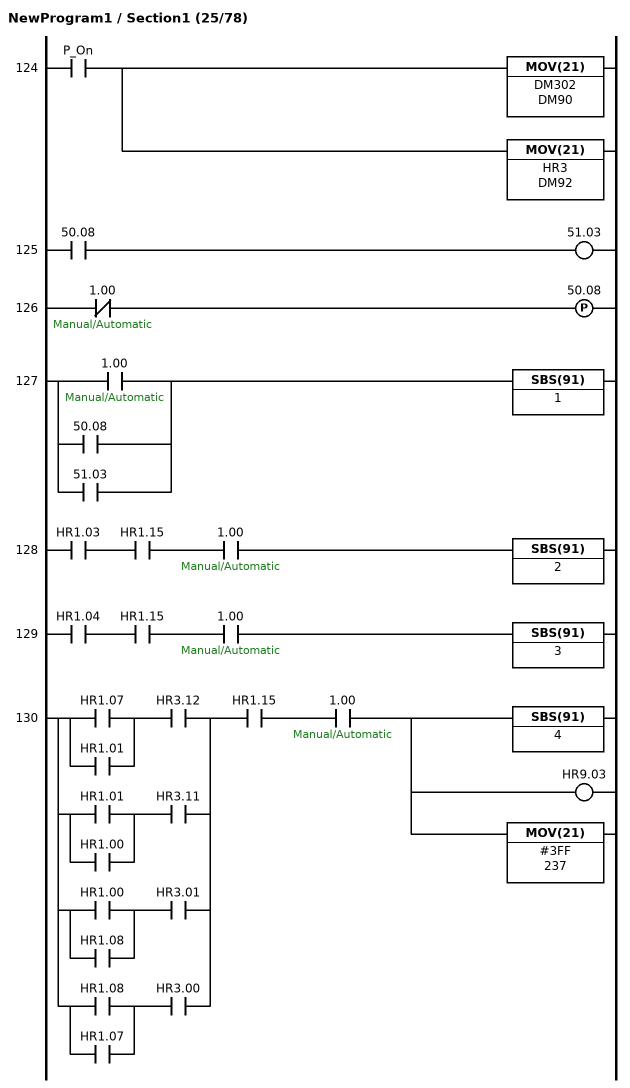
; [picture p24: NewProgram1 / Section1, rungs 124-130]
; rung 124
LD P_On
MOV(21) DM302 DM90
MOV(21) HR3 DM92
; rung 125
LD 50.08
OUT 51.03
; rung 126
LDNOT 1.00  ; Manual/Automatic
DIFU(13) 50.08
; rung 127
LD 1.00  ; Manual/Automatic
OR 50.08
OR 51.03
SBS(91) 1
; rung 128
LD HR1.03
AND HR1.15
AND 1.00  ; Manual/Automatic
SBS(91) 2
; rung 129
LD HR1.04
AND HR1.15
AND 1.00  ; Manual/Automatic
SBS(91) 3
; rung 130
LD HR1.07
OR HR1.01
AND HR3.12
LD HR1.01
OR HR1.00
AND HR3.11
ORLD
LD HR1.00
OR HR1.08
AND HR3.01
ORLD
LD HR1.08
OR HR1.07
AND HR3.00
ORLD
AND HR1.15
AND 1.00  ; Manual/Automatic
SBS(91) 4
OUT HR9.03
MOV(21) #3FF 237

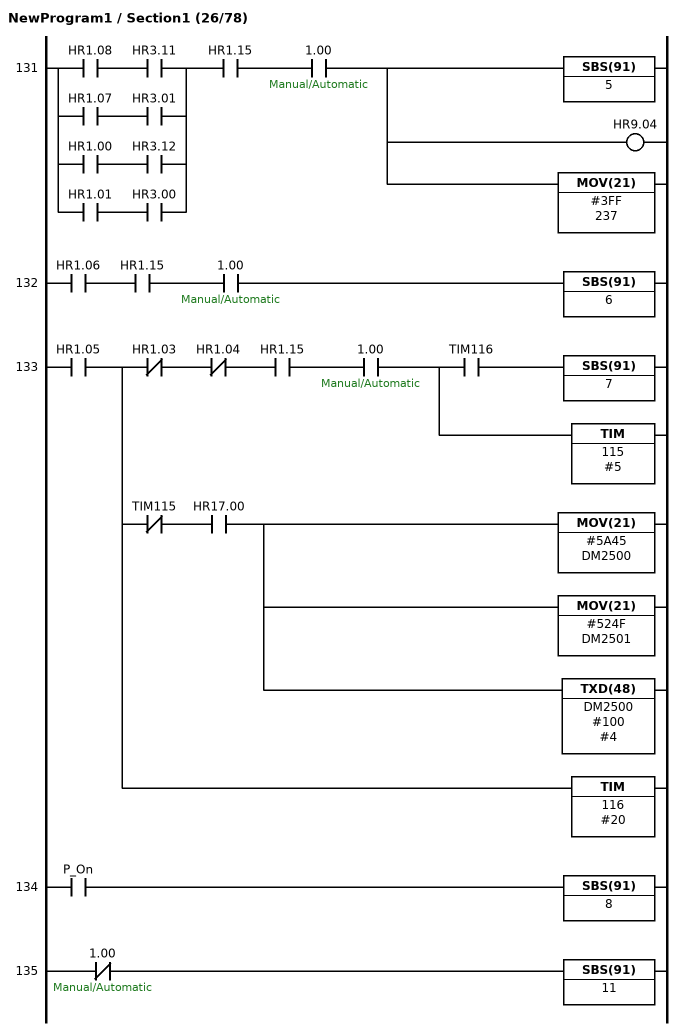
; rung 131
LD HR1.08
AND HR3.11
LD HR1.07
AND HR3.01
ORLD
LD HR1.00
AND HR3.12
ORLD
LD HR1.01
AND HR3.00
ORLD
AND HR1.15
AND 1.00  ; Manual/Automatic
SBS(91) 5
OUT HR9.04
MOV(21) #3FF 237
; rung 132
LD HR1.06
AND HR1.15
AND 1.00  ; Manual/Automatic
SBS(91) 6
; rung 133
LD HR1.05
OUT TR0
ANDNOT HR1.03
ANDNOT HR1.04
AND HR1.15
AND 1.00  ; Manual/Automatic
OUT TR1
AND TIM116
SBS(91) 7
LD TR1
TIM 115 #5
LD TR0
ANDNOT TIM115
AND HR17.00
MOV(21) #5A45 DM2500
MOV(21) #524F DM2501
TXD(48) DM2500 #100 #4
LD TR0
TIM 116 #20
; rung 134
LD P_On
SBS(91) 8
; rung 135
LDNOT 1.00  ; Manual/Automatic
SBS(91) 11

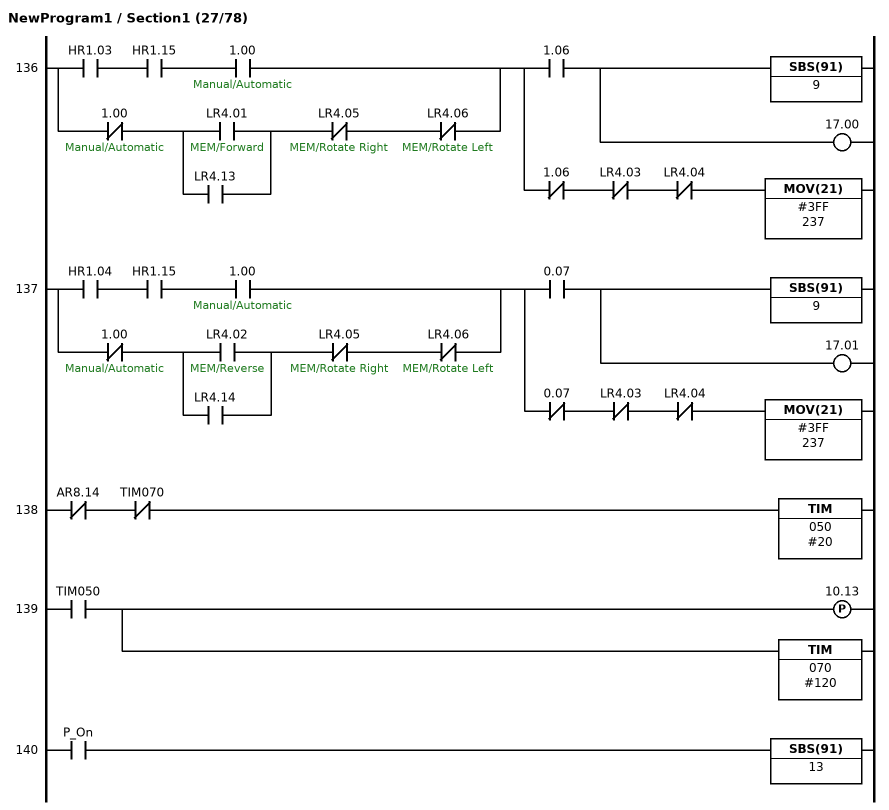
; rung 136
LD HR1.03
AND HR1.15
AND 1.00  ; Manual/Automatic
LDNOT 1.00  ; Manual/Automatic
LD LR4.01  ; MEM/Forward
OR LR4.13
ANDLD
ANDNOT LR4.05  ; MEM/Rotate Right
ANDNOT LR4.06  ; MEM/Rotate Left
ORLD
OUT TR0
AND 1.06
SBS(91) 9
OUT 17.00
LD TR0
ANDNOT 1.06
ANDNOT LR4.03
ANDNOT LR4.04
MOV(21) #3FF 237
; rung 137
LD HR1.04
AND HR1.15
AND 1.00  ; Manual/Automatic
LDNOT 1.00  ; Manual/Automatic
LD LR4.02  ; MEM/Reverse
OR LR4.14
ANDLD
ANDNOT LR4.05  ; MEM/Rotate Right
ANDNOT LR4.06  ; MEM/Rotate Left
ORLD
OUT TR0
AND 0.07
SBS(91) 9
OUT 17.01
LD TR0
ANDNOT 0.07
ANDNOT LR4.03
ANDNOT LR4.04
MOV(21) #3FF 237
; rung 138
LDNOT AR8.14
ANDNOT TIM070
TIM 050 #20
; rung 139
LD TIM050
DIFU(13) 10.13
TIM 070 #120
; rung 140
LD P_On
SBS(91) 13

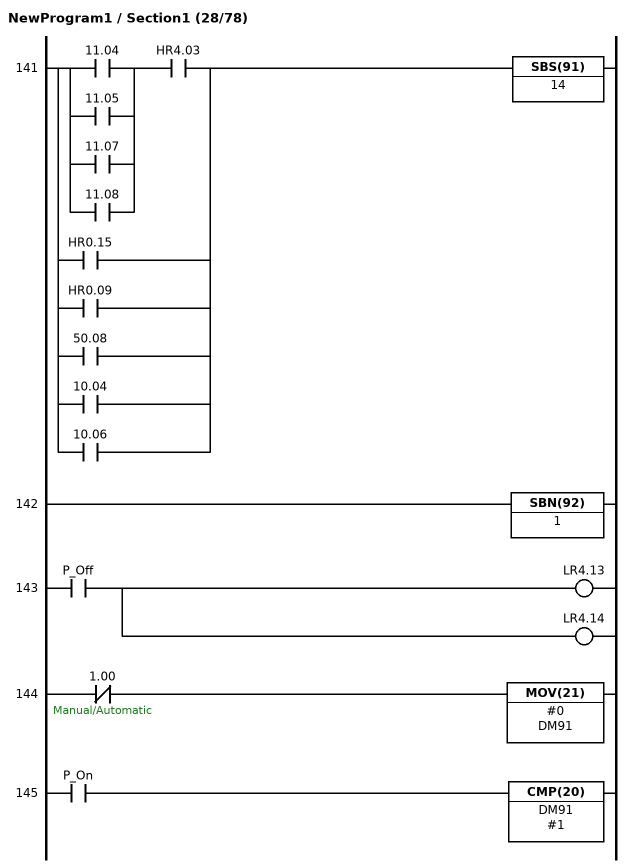
; rung 141
LD 11.04
OR 11.05
OR 11.07
OR 11.08
AND HR4.03
OR HR0.15
OR HR0.09
OR 50.08
OR 10.04
OR 10.06
SBS(91) 14
; rung 142
SBN(92) 1
; rung 143
LD P_Off
OUT LR4.13
OUT LR4.14
; rung 144
LDNOT 1.00  ; Manual/Automatic
MOV(21) #0 DM91
; rung 145
LD P_On
CMP(20) DM91 #1

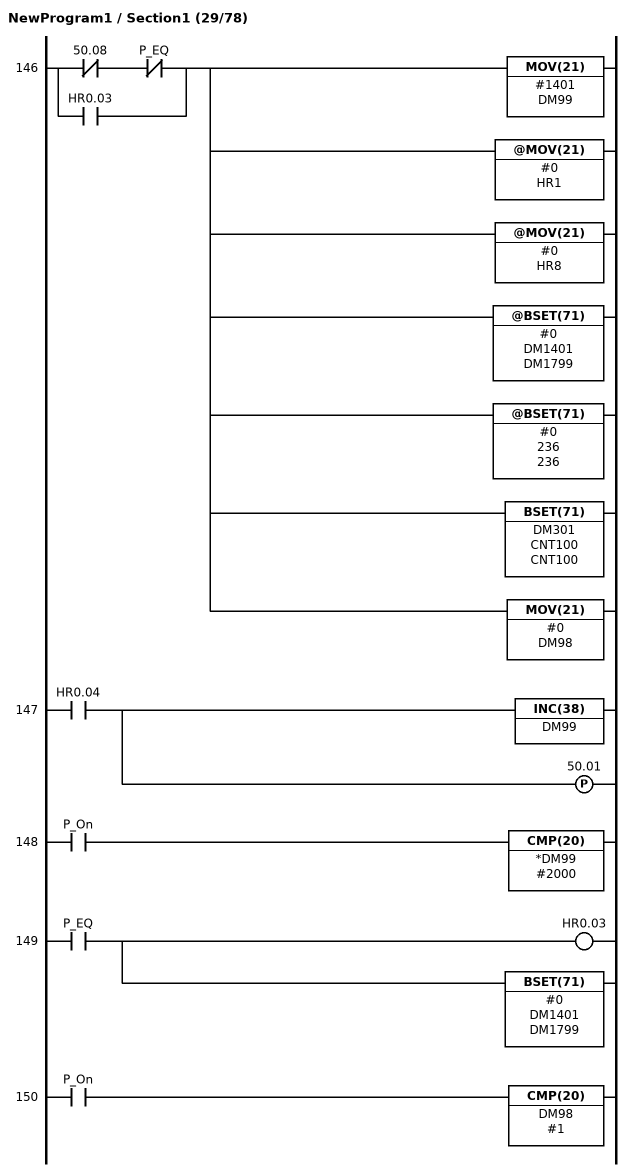
; rung 146
LDNOT 50.08
ANDNOT P_EQ
OR HR0.03
MOV(21) #1401 DM99
@MOV(21) #0 HR1
@MOV(21) #0 HR8
@BSET(71) #0 DM1401 DM1799
@BSET(71) #0 236 236
BSET(71) DM301 CNT100 CNT100
MOV(21) #0 DM98
; rung 147
LD HR0.04
INC(38) DM99
DIFU(13) 50.01
; rung 148
LD P_On
CMP(20) *DM99 #2000
; rung 149
LD P_EQ
OUT HR0.03
BSET(71) #0 DM1401 DM1799
; rung 150
LD P_On
CMP(20) DM98 #1

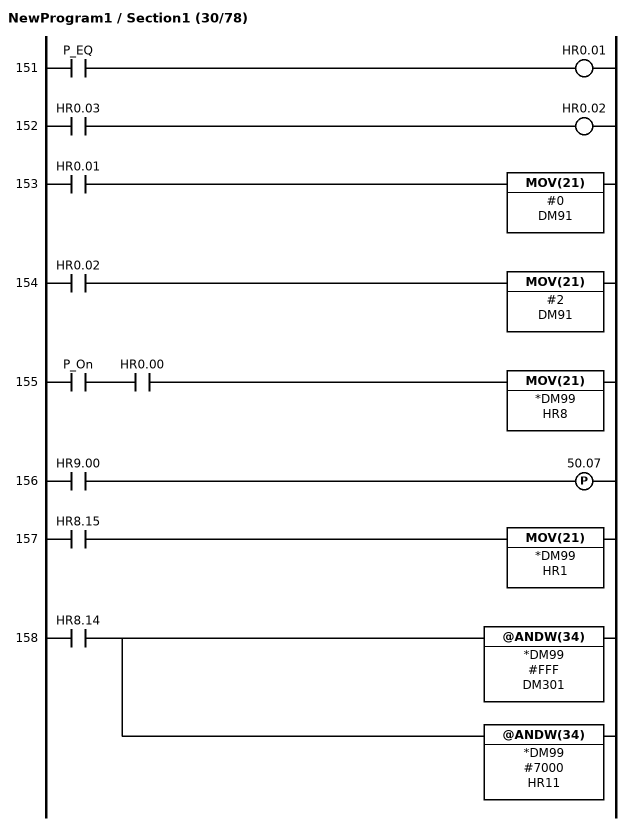
; rung 151
LD P_EQ
OUT HR0.01
; rung 152
LD HR0.03
OUT HR0.02
; rung 153
LD HR0.01
MOV(21) #0 DM91
; rung 154
LD HR0.02
MOV(21) #2 DM91
; rung 155
LD P_On
AND HR0.00
MOV(21) *DM99 HR8
; rung 156
LD HR9.00
DIFU(13) 50.07
; rung 157
LD HR8.15
MOV(21) *DM99 HR1
; rung 158
LD HR8.14
@ANDW(34) *DM99 #FFF DM301
@ANDW(34) *DM99 #7000 HR11

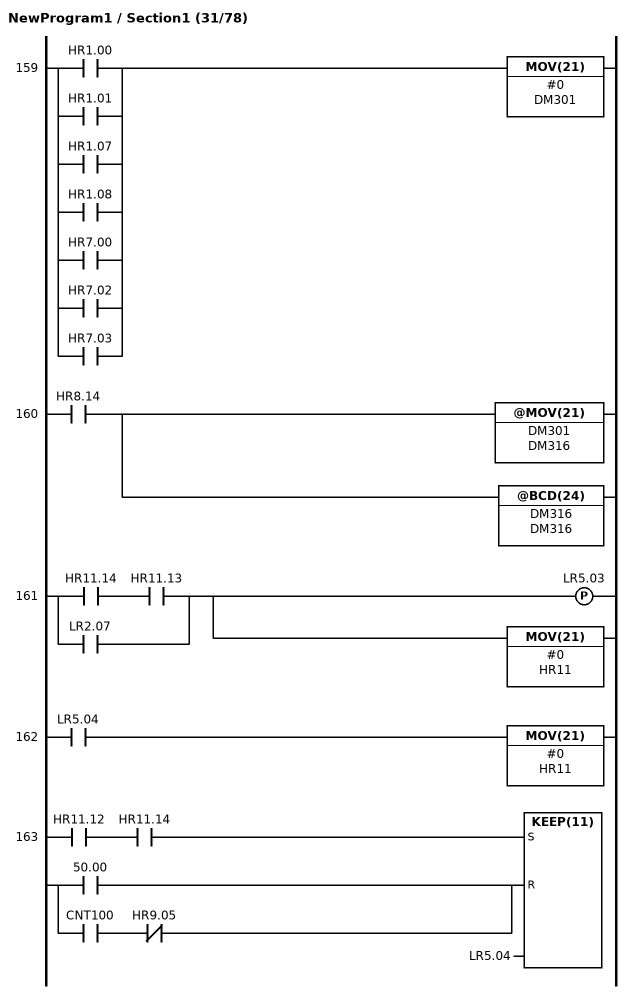
; rung 159
LD HR1.00
OR HR1.01
OR HR1.07
OR HR1.08
OR HR7.00
OR HR7.02
OR HR7.03
MOV(21) #0 DM301
; rung 160
LD HR8.14
@MOV(21) DM301 DM316
@BCD(24) DM316 DM316
; rung 161
LD HR11.14
AND HR11.13
OR LR2.07
DIFU(13) LR5.03
MOV(21) #0 HR11
; rung 162
LD LR5.04
MOV(21) #0 HR11
; rung 163
LD HR11.12
AND HR11.14
LD 50.00
LD CNT100
ANDNOT HR9.05
ORLD
KEEP(11) LR5.04

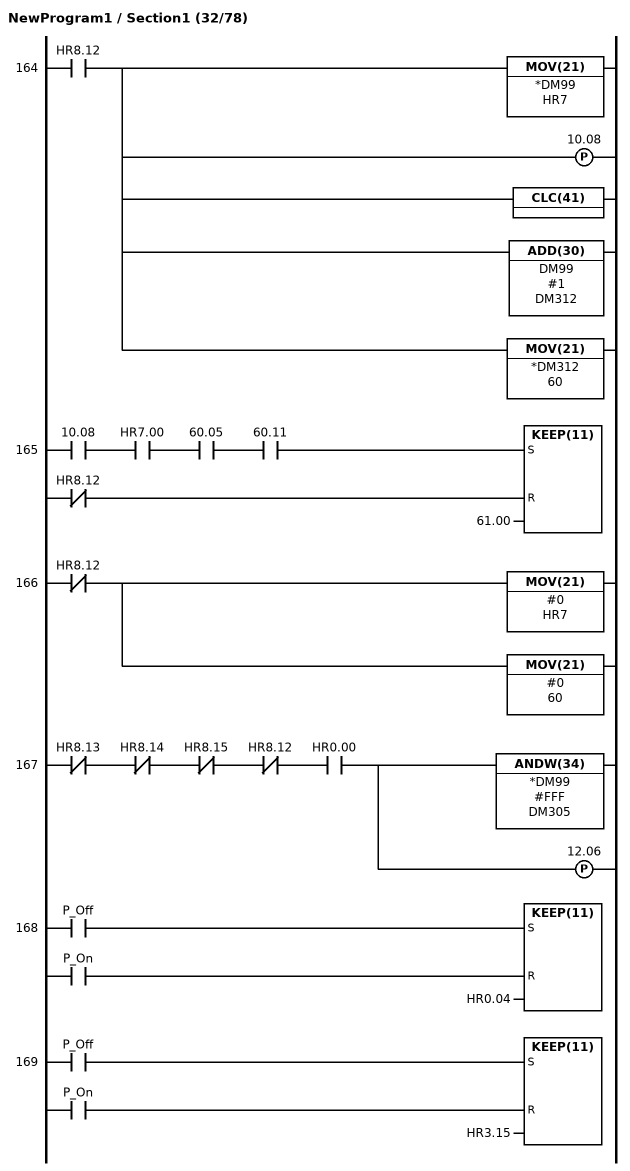
; rung 164
LD HR8.12
MOV(21) *DM99 HR7
DIFU(13) 10.08
CLC(41)
ADD(30) DM99 #1 DM312
MOV(21) *DM312 60
; rung 165
LD 10.08
AND HR7.00
AND 60.05
AND 60.11
LDNOT HR8.12
KEEP(11) 61.00
; rung 166
LDNOT HR8.12
MOV(21) #0 HR7
MOV(21) #0 60
; rung 167
LDNOT HR8.13
ANDNOT HR8.14
ANDNOT HR8.15
ANDNOT HR8.12
AND HR0.00
ANDW(34) *DM99 #FFF DM305
DIFU(13) 12.06
; rung 168
LD P_Off
LD P_On
KEEP(11) HR0.04
; rung 169
LD P_Off
LD P_On
KEEP(11) HR3.15

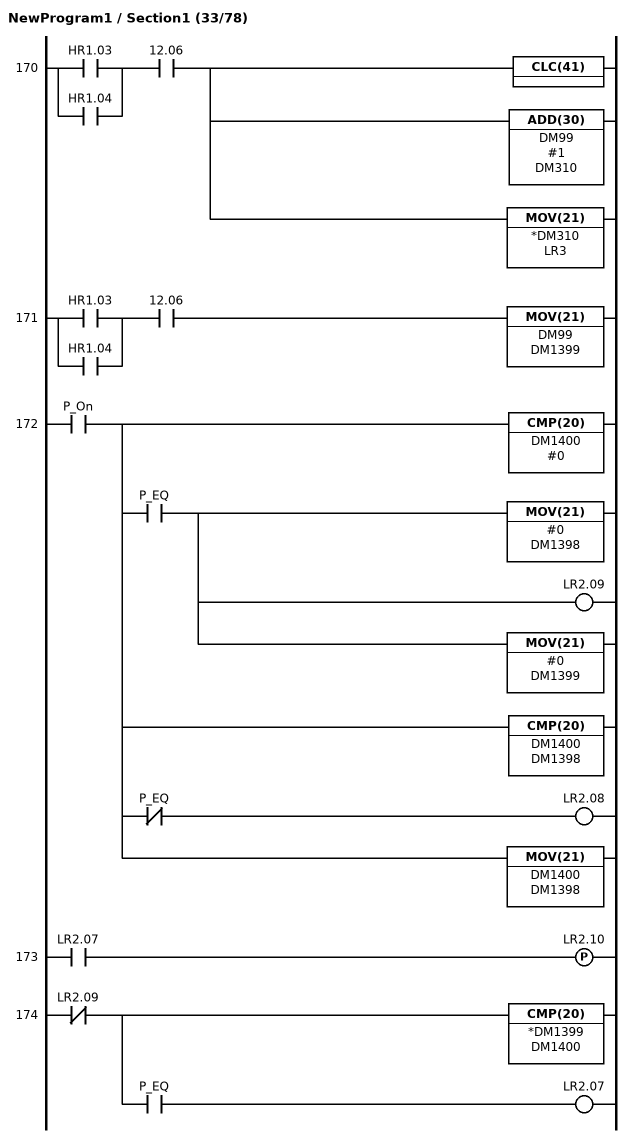
; rung 170
LD HR1.03
OR HR1.04
AND 12.06
CLC(41)
ADD(30) DM99 #1 DM310
MOV(21) *DM310 LR3
; rung 171
LD HR1.03
OR HR1.04
AND 12.06
MOV(21) DM99 DM1399
; rung 172
LD P_On
OUT TR0
CMP(20) DM1400 #0
AND P_EQ
MOV(21) #0 DM1398
OUT LR2.09
MOV(21) #0 DM1399
LD TR0
CMP(20) DM1400 DM1398
ANDNOT P_EQ
OUT LR2.08
LD TR0
MOV(21) DM1400 DM1398
; rung 173
LD LR2.07
DIFU(13) LR2.10
; rung 174
LDNOT LR2.09
CMP(20) *DM1399 DM1400
AND P_EQ
OUT LR2.07

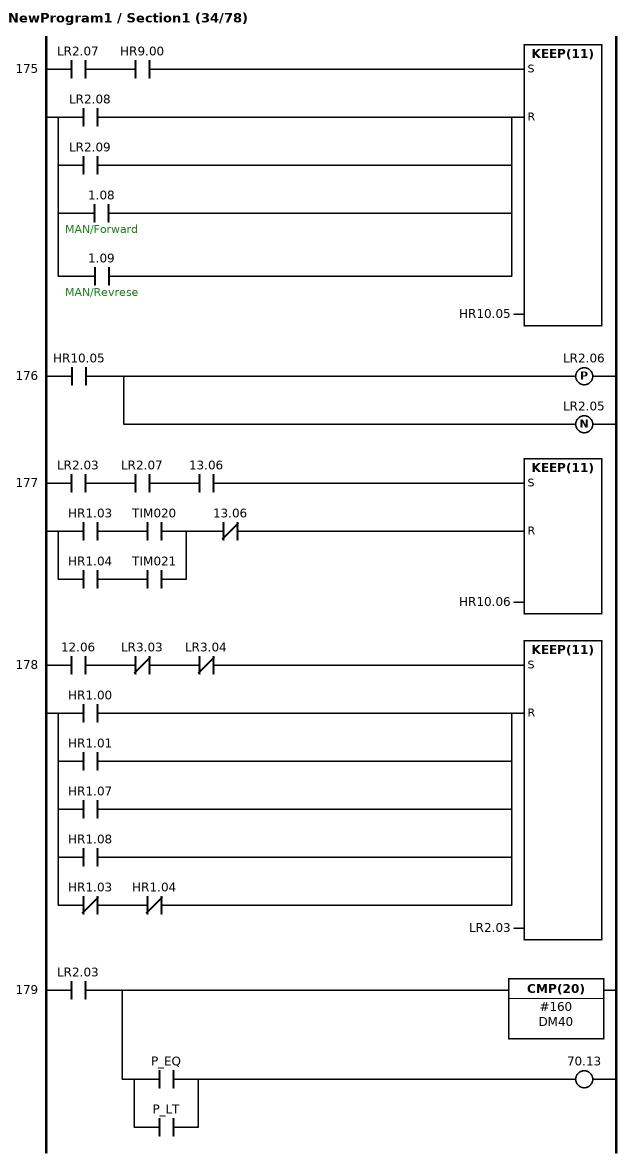
; rung 175
LD LR2.07
AND HR9.00
LD LR2.08
OR LR2.09
OR 1.08  ; MAN/Forward
OR 1.09  ; MAN/Revrese
KEEP(11) HR10.05
; rung 176
LD HR10.05
DIFU(13) LR2.06
DIFD(14) LR2.05
; rung 177
LD LR2.03
AND LR2.07
AND 13.06
LD HR1.03
AND TIM020
LD HR1.04
AND TIM021
ORLD
ANDNOT 13.06
KEEP(11) HR10.06
; rung 178
LD 12.06
ANDNOT LR3.03
ANDNOT LR3.04
LD HR1.00
OR HR1.01
OR HR1.07
OR HR1.08
LDNOT HR1.03
ANDNOT HR1.04
ORLD
KEEP(11) LR2.03
; rung 179
LD LR2.03
CMP(20) #160 DM40
LD P_EQ
OR P_LT
ANDLD
OUT 70.13

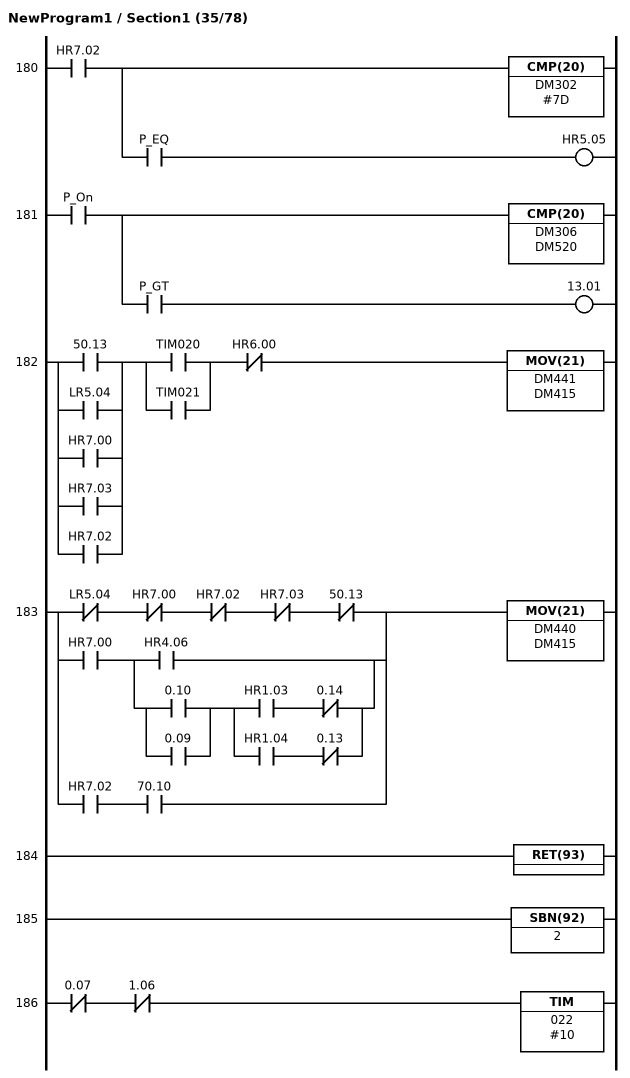
; rung 180
LD HR7.02
CMP(20) DM302 #7D
AND P_EQ
OUT HR5.05
; rung 181
LD P_On
CMP(20) DM306 DM520
AND P_GT
OUT 13.01
; rung 182
LD 50.13
OR LR5.04
OR HR7.00
OR HR7.03
OR HR7.02
LD TIM020
OR TIM021
ANDLD
ANDNOT HR6.00
MOV(21) DM441 DM415
; rung 183
LDNOT LR5.04
ANDNOT HR7.00
ANDNOT HR7.02
ANDNOT HR7.03
ANDNOT 50.13
LD HR7.00
LD HR4.06
LD 0.10
OR 0.09
LD HR1.03
ANDNOT 0.14
LD HR1.04
ANDNOT 0.13
ORLD
ANDLD
ORLD
ANDLD
ORLD
LD HR7.02
AND 70.10
ORLD
MOV(21) DM440 DM415
; rung 184
RET(93)
; rung 185
SBN(92) 2
; rung 186
LDNOT 0.07
ANDNOT 1.06
TIM 022 #10

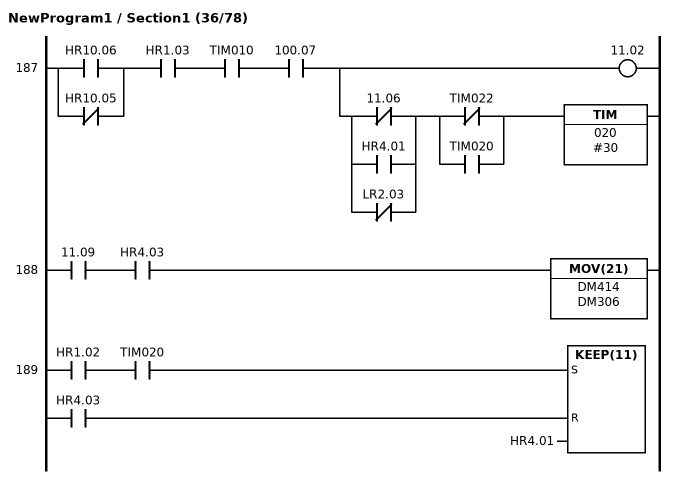
; rung 187
LD HR10.06
ORNOT HR10.05
AND HR1.03
AND TIM010
AND 100.07
OUT 11.02
LDNOT 11.06
OR HR4.01
ORNOT LR2.03
ANDLD
LDNOT TIM022
OR TIM020
ANDLD
TIM 020 #30
; rung 188
LD 11.09
AND HR4.03
MOV(21) DM414 DM306
; rung 189
LD HR1.02
AND TIM020
LD HR4.03
KEEP(11) HR4.01

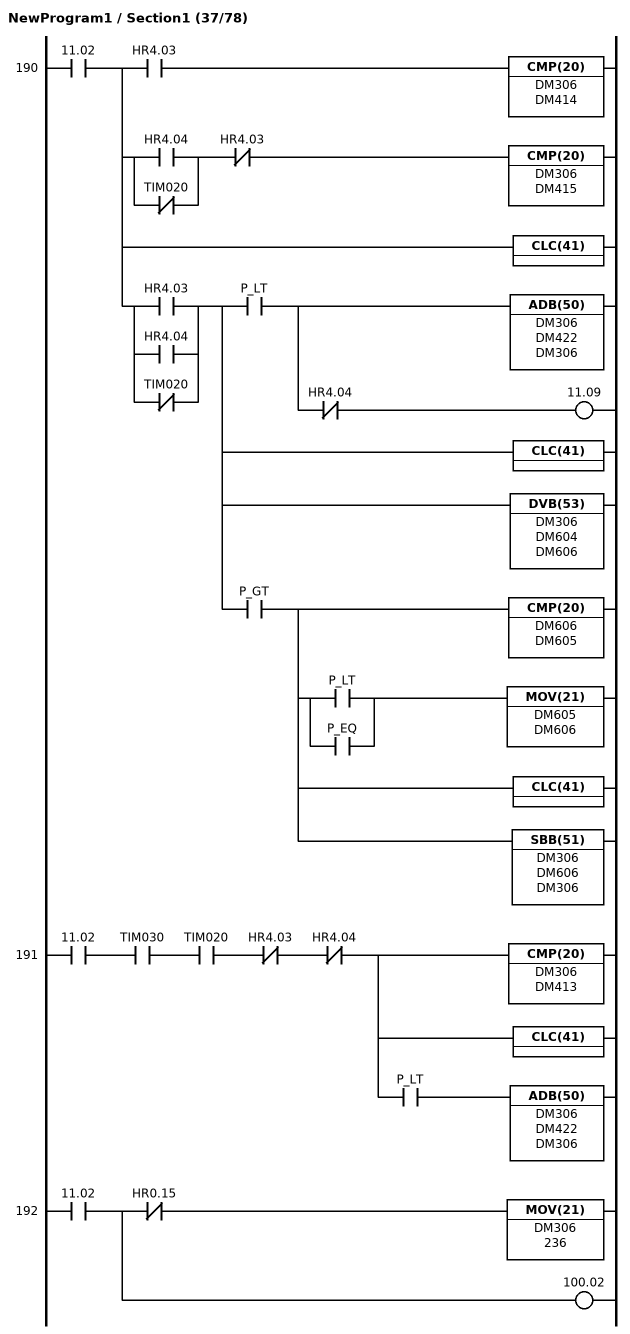
; rung 190
LD 11.02
OUT TR0
AND HR4.03
CMP(20) DM306 DM414
LD TR0
LD HR4.04
ORNOT TIM020
ANDLD
ANDNOT HR4.03
CMP(20) DM306 DM415
LD TR0
CLC(41)
LD HR4.03
OR HR4.04
ORNOT TIM020
ANDLD
OUT TR0
AND P_LT
ADB(50) DM306 DM422 DM306
ANDNOT HR4.04
OUT 11.09
LD TR0
CLC(41)
DVB(53) DM306 DM604 DM606
AND P_GT
OUT TR0
CMP(20) DM606 DM605
LD P_LT
OR P_EQ
ANDLD
MOV(21) DM605 DM606
LD TR0
CLC(41)
SBB(51) DM306 DM606 DM306
; rung 191
LD 11.02
AND TIM030
AND TIM020
ANDNOT HR4.03
ANDNOT HR4.04
CMP(20) DM306 DM413
CLC(41)
AND P_LT
ADB(50) DM306 DM422 DM306
; rung 192
LD 11.02
OUT TR0
ANDNOT HR0.15
MOV(21) DM306 236
LD TR0
OUT 100.02

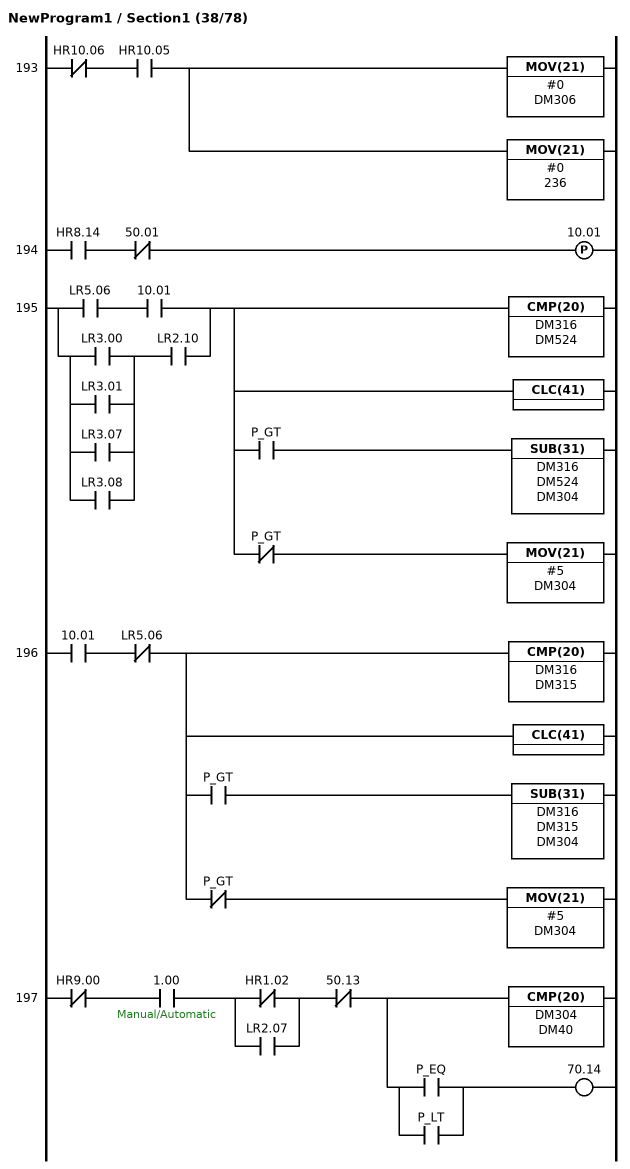
; rung 193
LDNOT HR10.06
AND HR10.05
MOV(21) #0 DM306
MOV(21) #0 236
; rung 194
LD HR8.14
ANDNOT 50.01
DIFU(13) 10.01
; rung 195
LD LR5.06
AND 10.01
LD LR3.00
OR LR3.01
OR LR3.07
OR LR3.08
AND LR2.10
ORLD
OUT TR0
CMP(20) DM316 DM524
CLC(41)
AND P_GT
SUB(31) DM316 DM524 DM304
LD TR0
ANDNOT P_GT
MOV(21) #5 DM304
; rung 196
LD 10.01
ANDNOT LR5.06
OUT TR0
CMP(20) DM316 DM315
CLC(41)
AND P_GT
SUB(31) DM316 DM315 DM304
LD TR0
ANDNOT P_GT
MOV(21) #5 DM304
; rung 197
LDNOT HR9.00
AND 1.00  ; Manual/Automatic
LDNOT HR1.02
OR LR2.07
ANDLD
ANDNOT 50.13
CMP(20) DM304 DM40
LD P_EQ
OR P_LT
ANDLD
OUT 70.14

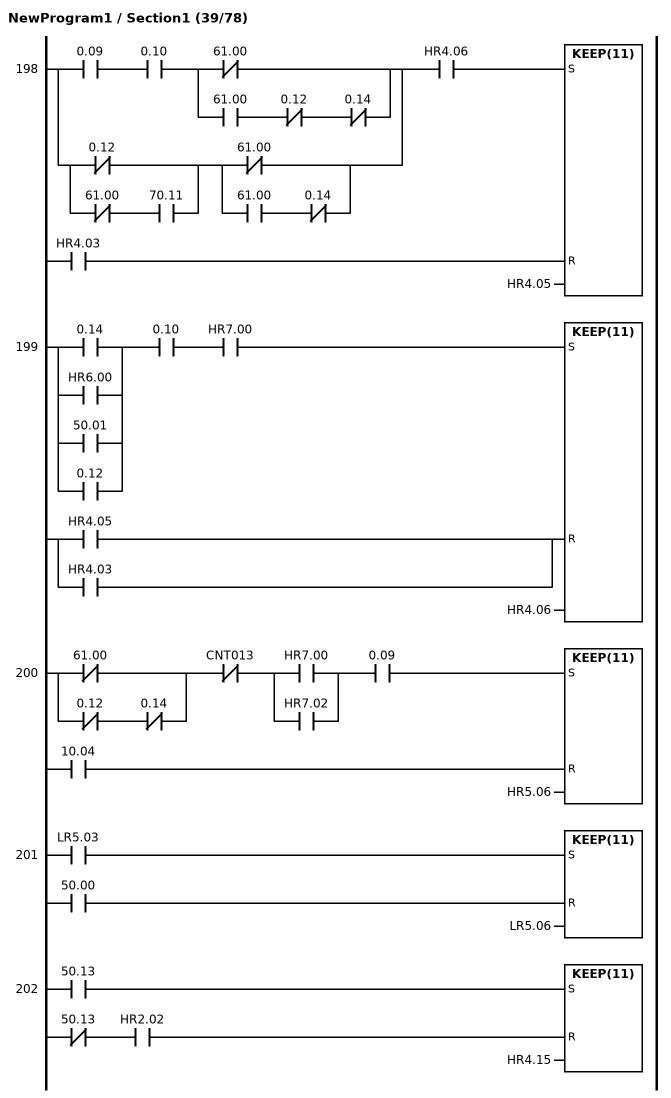
; rung 198
LD 0.09
AND 0.10
LDNOT 61.00
LD 61.00
ANDNOT 0.12
ANDNOT 0.14
ORLD
ANDLD
LDNOT 0.12
LDNOT 61.00
AND 70.11
ORLD
LDNOT 61.00
LD 61.00
ANDNOT 0.14
ORLD
ANDLD
ORLD
AND HR4.06
LD HR4.03
KEEP(11) HR4.05
; rung 199
LD 0.14
OR HR6.00
OR 50.01
OR 0.12
AND 0.10
AND HR7.00
LD HR4.05
OR HR4.03
KEEP(11) HR4.06
; rung 200
LDNOT 61.00
LDNOT 0.12
ANDNOT 0.14
ORLD
ANDNOT CNT013
LD HR7.00
OR HR7.02
ANDLD
AND 0.09
LD 10.04
KEEP(11) HR5.06
; rung 201
LD LR5.03
LD 50.00
KEEP(11) LR5.06
; rung 202
LD 50.13
LDNOT 50.13
AND HR2.02
KEEP(11) HR4.15

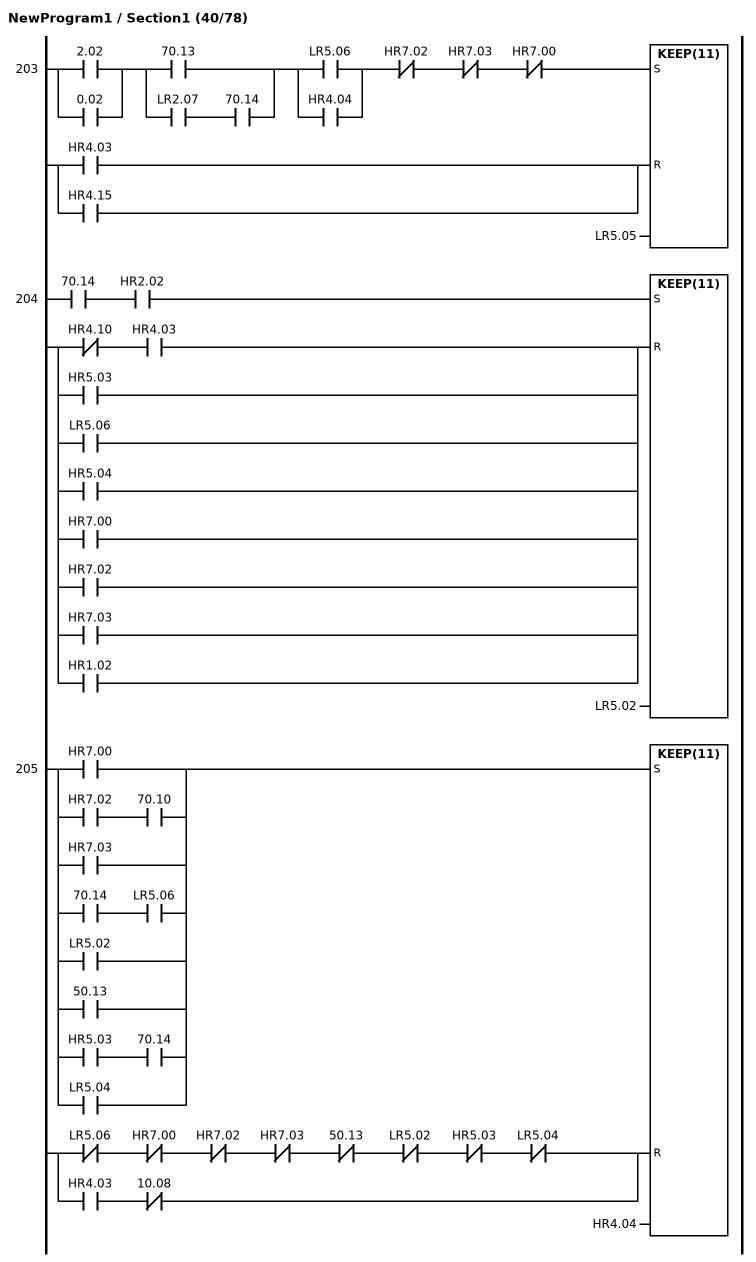
; rung 203
LD 2.02
OR 0.02
LD 70.13
LD LR2.07
AND 70.14
ORLD
ANDLD
LD LR5.06
OR HR4.04
ANDLD
ANDNOT HR7.02
ANDNOT HR7.03
ANDNOT HR7.00
LD HR4.03
OR HR4.15
KEEP(11) LR5.05
; rung 204
LD 70.14
AND HR2.02
LDNOT HR4.10
AND HR4.03
OR HR5.03
OR LR5.06
OR HR5.04
OR HR7.00
OR HR7.02
OR HR7.03
OR HR1.02
KEEP(11) LR5.02
; rung 205
LD HR7.00
LD HR7.02
AND 70.10
ORLD
OR HR7.03
LD 70.14
AND LR5.06
ORLD
OR LR5.02
OR 50.13
LD HR5.03
AND 70.14
ORLD
OR LR5.04
LDNOT LR5.06
ANDNOT HR7.00
ANDNOT HR7.02
ANDNOT HR7.03
ANDNOT 50.13
ANDNOT LR5.02
ANDNOT HR5.03
ANDNOT LR5.04
LD HR4.03
ANDNOT 10.08
ORLD
KEEP(11) HR4.04

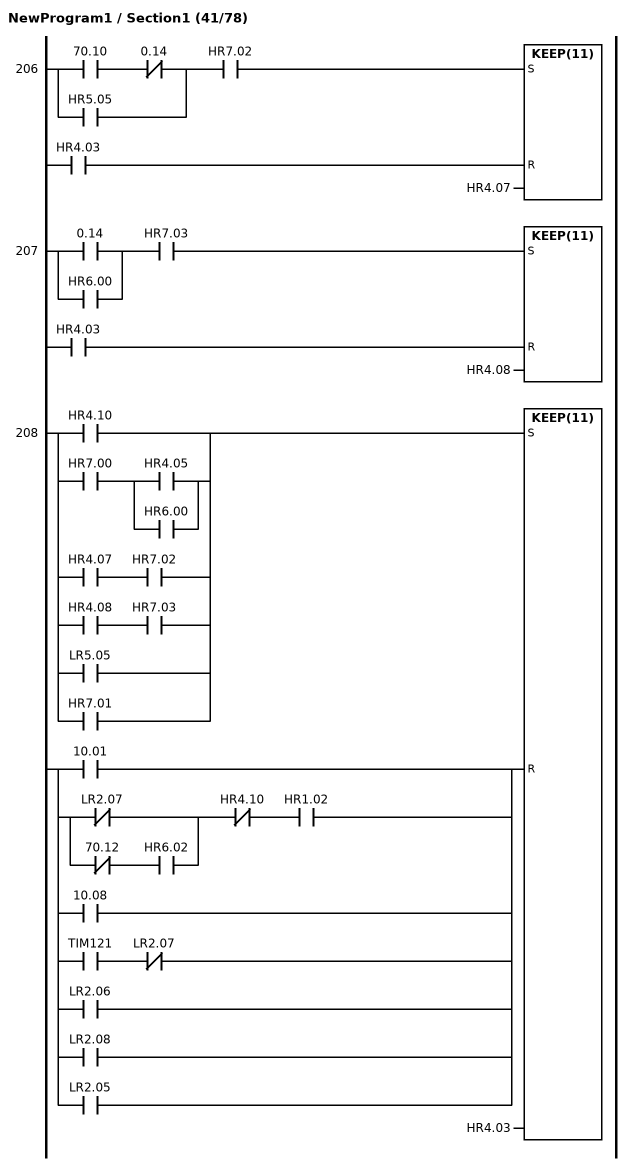
; rung 206
LD 70.10
ANDNOT 0.14
OR HR5.05
AND HR7.02
LD HR4.03
KEEP(11) HR4.07
; rung 207
LD 0.14
OR HR6.00
AND HR7.03
LD HR4.03
KEEP(11) HR4.08
; rung 208
LD HR4.10
LD HR7.00
LD HR4.05
OR HR6.00
ANDLD
ORLD
LD HR4.07
AND HR7.02
ORLD
LD HR4.08
AND HR7.03
ORLD
OR LR5.05
OR HR7.01
LD 10.01
LDNOT LR2.07
LDNOT 70.12
AND HR6.02
ORLD
ANDNOT HR4.10
AND HR1.02
ORLD
OR 10.08
LD TIM121
ANDNOT LR2.07
ORLD
OR LR2.06
OR LR2.08
OR LR2.05
KEEP(11) HR4.03

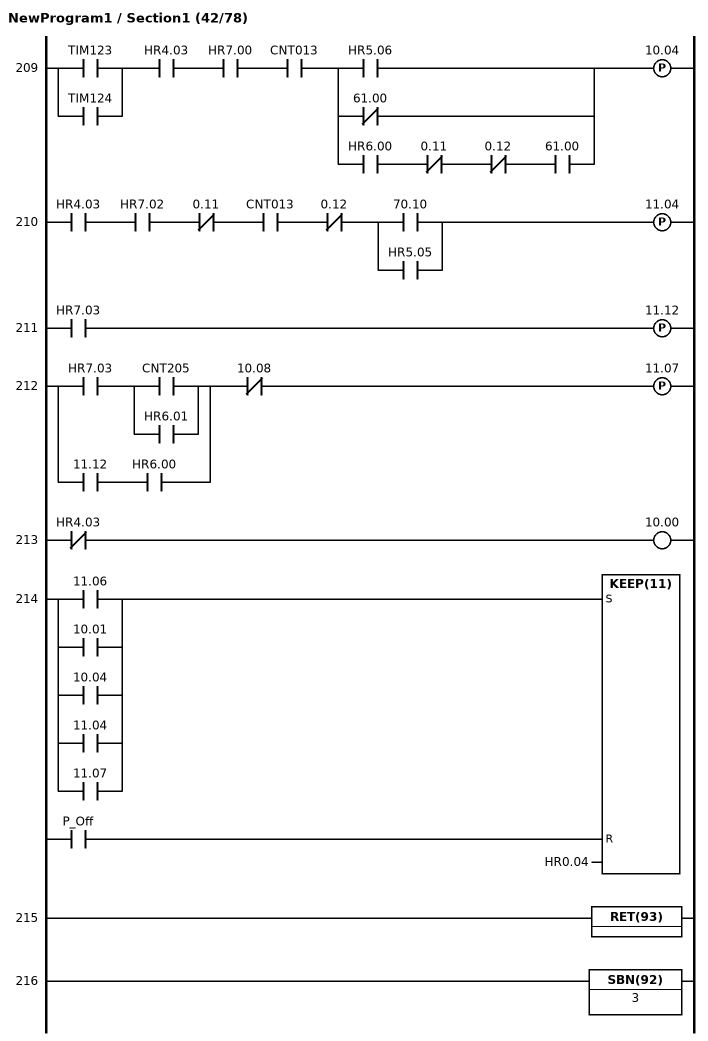
; rung 209
LD TIM123
OR TIM124
AND HR4.03
AND HR7.00
AND CNT013
LD HR5.06
ORNOT 61.00
LD HR6.00
ANDNOT 0.11
ANDNOT 0.12
AND 61.00
ORLD
ANDLD
DIFU(13) 10.04
; rung 210
LD HR4.03
AND HR7.02
ANDNOT 0.11
AND CNT013
ANDNOT 0.12
LD 70.10
OR HR5.05
ANDLD
DIFU(13) 11.04
; rung 211
LD HR7.03
DIFU(13) 11.12
; rung 212
LD HR7.03
LD CNT205
OR HR6.01
ANDLD
LD 11.12
AND HR6.00
ORLD
ANDNOT 10.08
DIFU(13) 11.07
; rung 213
LDNOT HR4.03
OUT 10.00
; rung 214
LD 11.06
OR 10.01
OR 10.04
OR 11.04
OR 11.07
LD P_Off
KEEP(11) HR0.04
; rung 215
RET(93)
; rung 216
SBN(92) 3

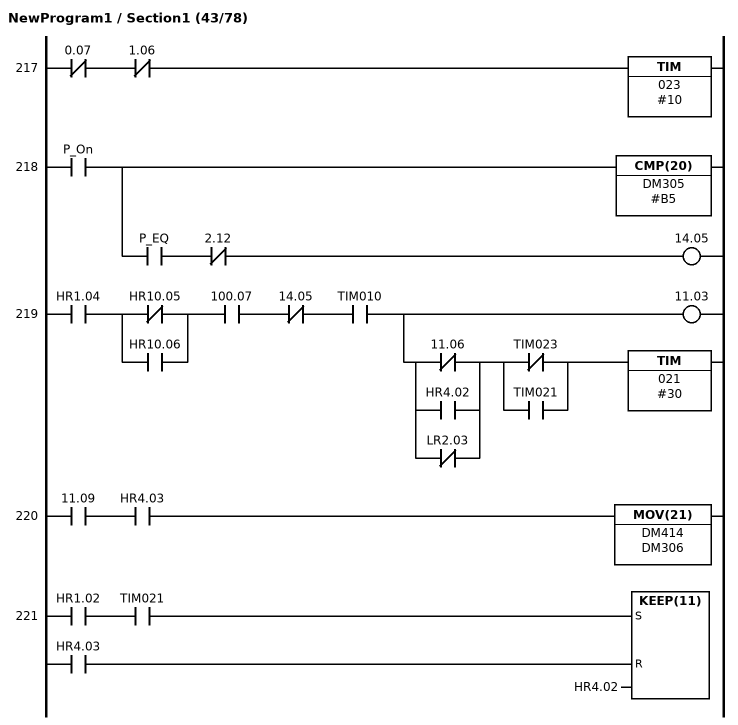
; rung 217
LDNOT 0.07
ANDNOT 1.06
TIM 023 #10
; rung 218
LD P_On
CMP(20) DM305 #B5
AND P_EQ
ANDNOT 2.12
OUT 14.05
; rung 219
LD HR1.04
LDNOT HR10.05
OR HR10.06
ANDLD
AND 100.07
ANDNOT 14.05
AND TIM010
OUT 11.03
LDNOT 11.06
OR HR4.02
ORNOT LR2.03
ANDLD
LDNOT TIM023
OR TIM021
ANDLD
TIM 021 #30
; rung 220
LD 11.09
AND HR4.03
MOV(21) DM414 DM306
; rung 221
LD HR1.02
AND TIM021
LD HR4.03
KEEP(11) HR4.02

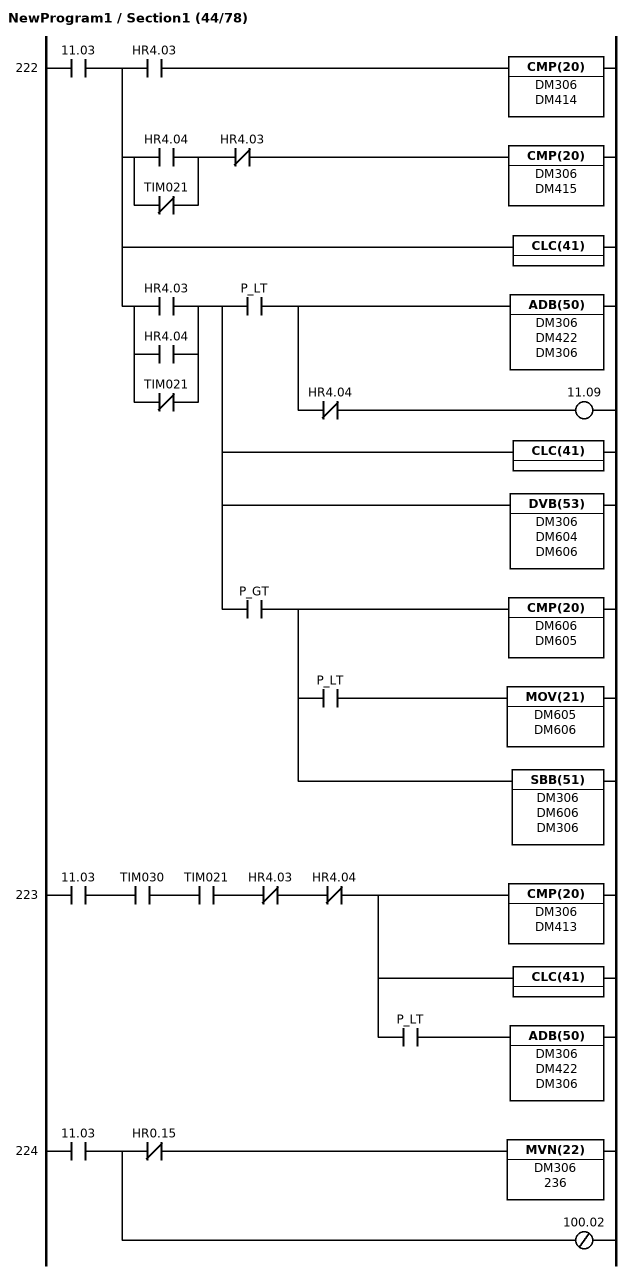
; rung 222
LD 11.03
OUT TR0
AND HR4.03
CMP(20) DM306 DM414
LD TR0
LD HR4.04
ORNOT TIM021
ANDLD
ANDNOT HR4.03
CMP(20) DM306 DM415
LD TR0
CLC(41)
LD HR4.03
OR HR4.04
ORNOT TIM021
ANDLD
OUT TR0
AND P_LT
ADB(50) DM306 DM422 DM306
ANDNOT HR4.04
OUT 11.09
LD TR0
CLC(41)
DVB(53) DM306 DM604 DM606
AND P_GT
OUT TR0
CMP(20) DM606 DM605
AND P_LT
MOV(21) DM605 DM606
LD TR0
SBB(51) DM306 DM606 DM306
; rung 223
LD 11.03
AND TIM030
AND TIM021
ANDNOT HR4.03
ANDNOT HR4.04
CMP(20) DM306 DM413
CLC(41)
AND P_LT
ADB(50) DM306 DM422 DM306
; rung 224
LD 11.03
OUT TR0
ANDNOT HR0.15
MVN(22) DM306 236
LD TR0
OUTNOT 100.02

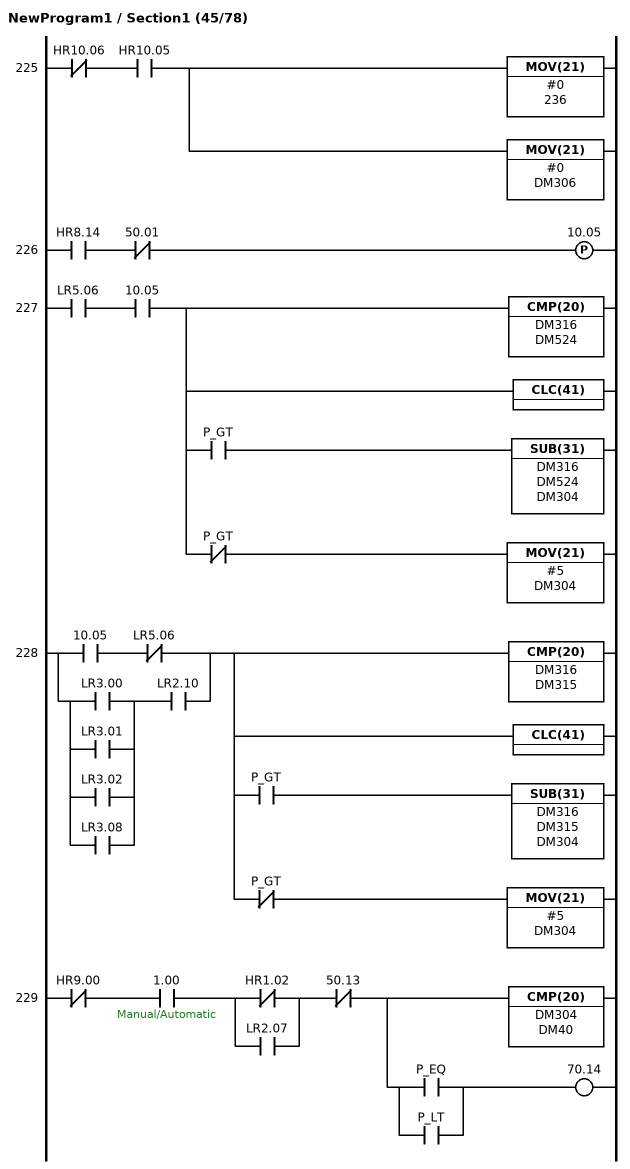
; rung 225
LDNOT HR10.06
AND HR10.05
MOV(21) #0 236
MOV(21) #0 DM306
; rung 226
LD HR8.14
ANDNOT 50.01
DIFU(13) 10.05
; rung 227
LD LR5.06
AND 10.05
OUT TR0
CMP(20) DM316 DM524
CLC(41)
AND P_GT
SUB(31) DM316 DM524 DM304
LD TR0
ANDNOT P_GT
MOV(21) #5 DM304
; rung 228
LD 10.05
ANDNOT LR5.06
LD LR3.00
OR LR3.01
OR LR3.02
OR LR3.08
AND LR2.10
ORLD
OUT TR0
CMP(20) DM316 DM315
CLC(41)
AND P_GT
SUB(31) DM316 DM315 DM304
LD TR0
ANDNOT P_GT
MOV(21) #5 DM304
; rung 229
LDNOT HR9.00
AND 1.00  ; Manual/Automatic
LDNOT HR1.02
OR LR2.07
ANDLD
ANDNOT 50.13
CMP(20) DM304 DM40
LD P_EQ
OR P_LT
ANDLD
OUT 70.14

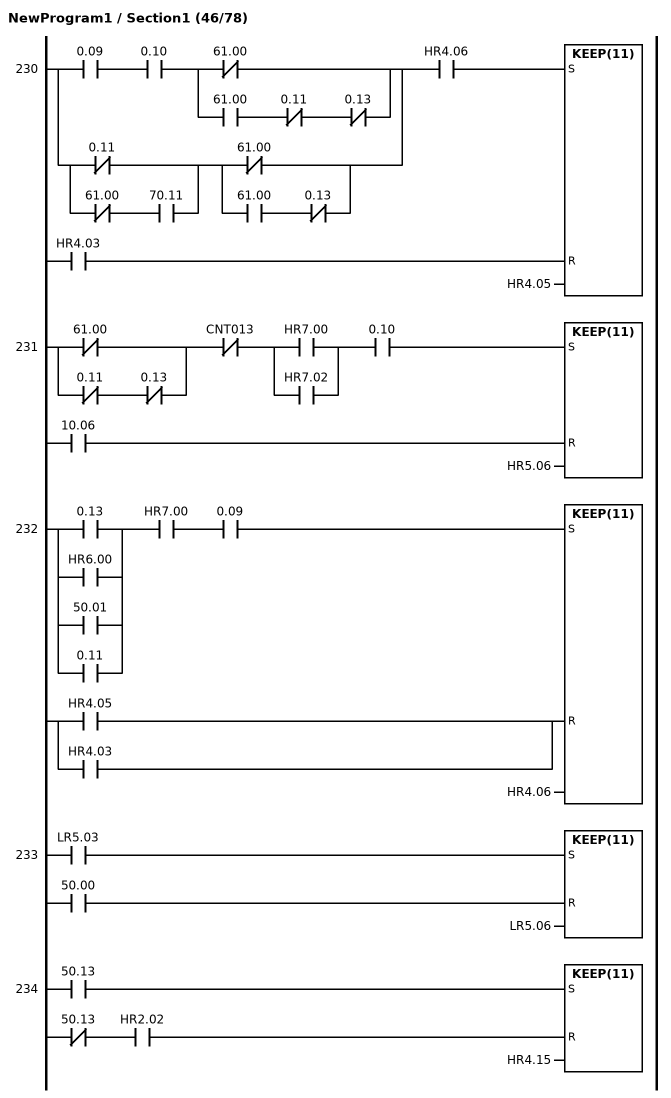
; rung 230
LD 0.09
AND 0.10
LDNOT 61.00
LD 61.00
ANDNOT 0.11
ANDNOT 0.13
ORLD
ANDLD
LDNOT 0.11
LDNOT 61.00
AND 70.11
ORLD
LDNOT 61.00
LD 61.00
ANDNOT 0.13
ORLD
ANDLD
ORLD
AND HR4.06
LD HR4.03
KEEP(11) HR4.05
; rung 231
LDNOT 61.00
LDNOT 0.11
ANDNOT 0.13
ORLD
ANDNOT CNT013
LD HR7.00
OR HR7.02
ANDLD
AND 0.10
LD 10.06
KEEP(11) HR5.06
; rung 232
LD 0.13
OR HR6.00
OR 50.01
OR 0.11
AND HR7.00
AND 0.09
LD HR4.05
OR HR4.03
KEEP(11) HR4.06
; rung 233
LD LR5.03
LD 50.00
KEEP(11) LR5.06
; rung 234
LD 50.13
LDNOT 50.13
AND HR2.02
KEEP(11) HR4.15

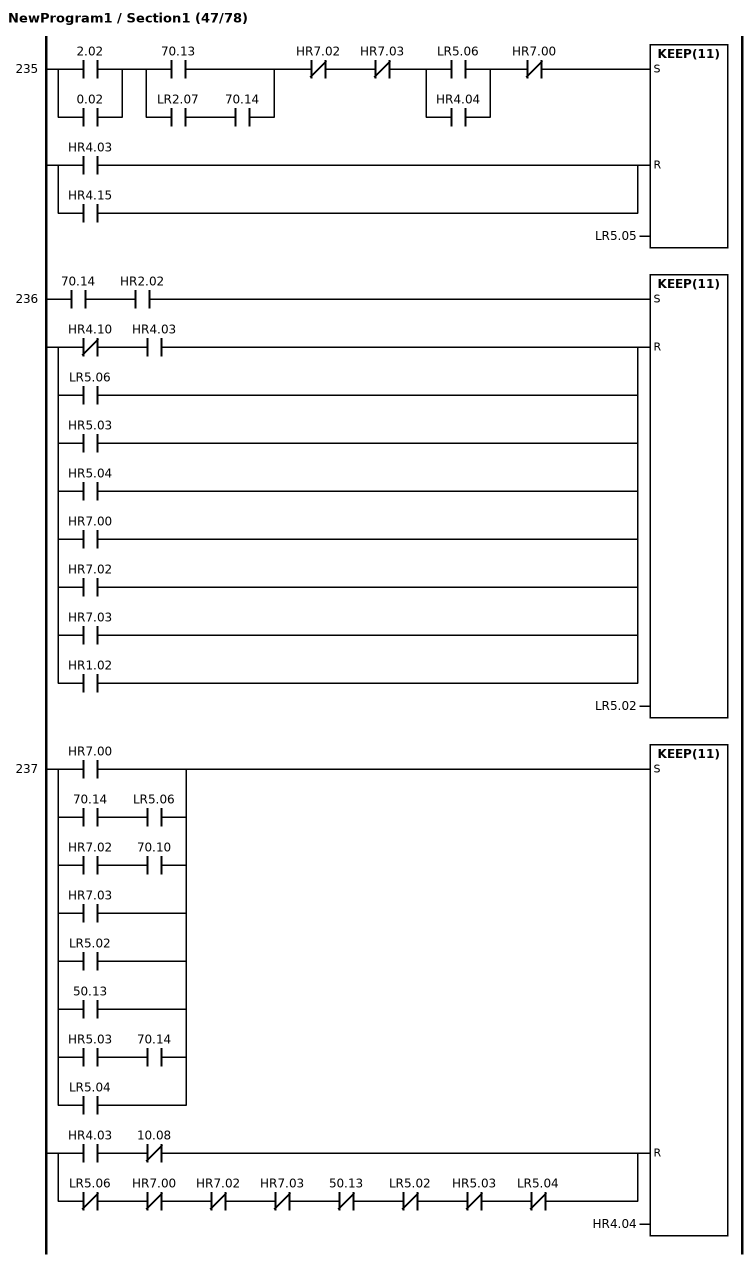
; rung 235
LD 2.02
OR 0.02
LD 70.13
LD LR2.07
AND 70.14
ORLD
ANDLD
ANDNOT HR7.02
ANDNOT HR7.03
LD LR5.06
OR HR4.04
ANDLD
ANDNOT HR7.00
LD HR4.03
OR HR4.15
KEEP(11) LR5.05
; rung 236
LD 70.14
AND HR2.02
LDNOT HR4.10
AND HR4.03
OR LR5.06
OR HR5.03
OR HR5.04
OR HR7.00
OR HR7.02
OR HR7.03
OR HR1.02
KEEP(11) LR5.02
; rung 237
LD HR7.00
LD 70.14
AND LR5.06
ORLD
LD HR7.02
AND 70.10
ORLD
OR HR7.03
OR LR5.02
OR 50.13
LD HR5.03
AND 70.14
ORLD
OR LR5.04
LD HR4.03
ANDNOT 10.08
LDNOT LR5.06
ANDNOT HR7.00
ANDNOT HR7.02
ANDNOT HR7.03
ANDNOT 50.13
ANDNOT LR5.02
ANDNOT HR5.03
ANDNOT LR5.04
ORLD
KEEP(11) HR4.04

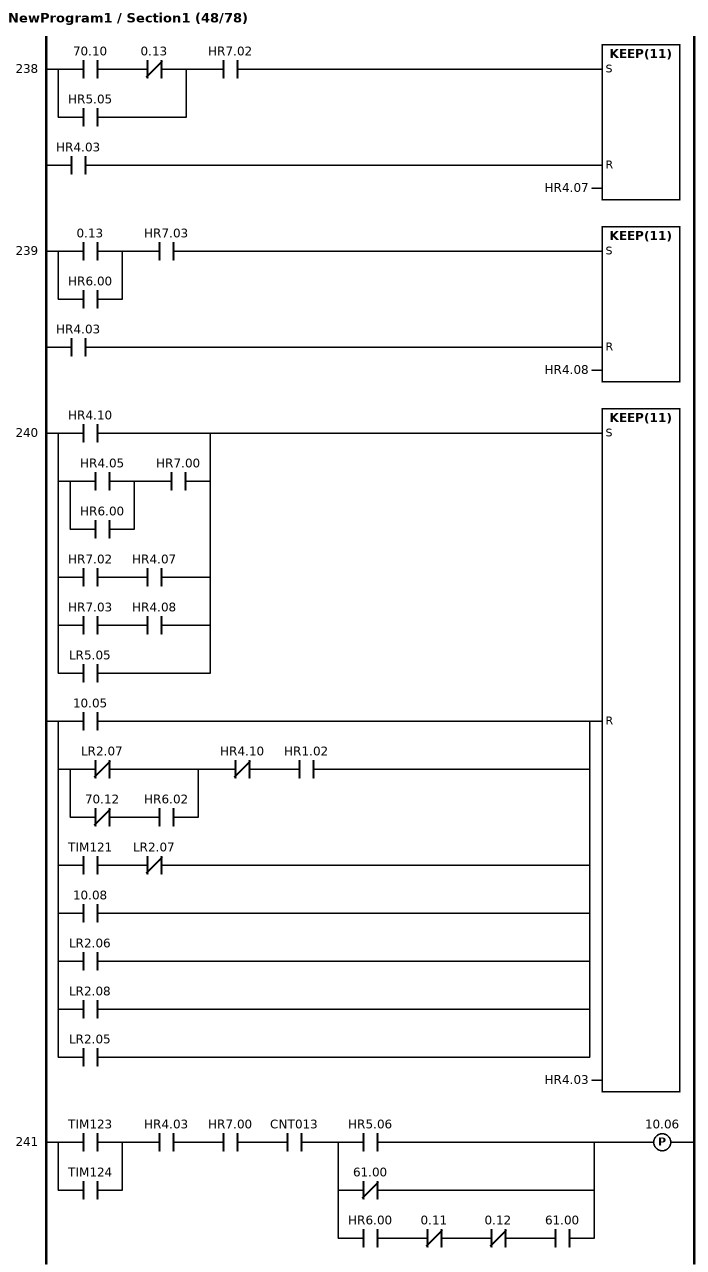
; rung 238
LD 70.10
ANDNOT 0.13
OR HR5.05
AND HR7.02
LD HR4.03
KEEP(11) HR4.07
; rung 239
LD 0.13
OR HR6.00
AND HR7.03
LD HR4.03
KEEP(11) HR4.08
; rung 240
LD HR4.10
LD HR4.05
OR HR6.00
AND HR7.00
ORLD
LD HR7.02
AND HR4.07
ORLD
LD HR7.03
AND HR4.08
ORLD
OR LR5.05
LD 10.05
LDNOT LR2.07
LDNOT 70.12
AND HR6.02
ORLD
ANDNOT HR4.10
AND HR1.02
ORLD
LD TIM121
ANDNOT LR2.07
ORLD
OR 10.08
OR LR2.06
OR LR2.08
OR LR2.05
KEEP(11) HR4.03
; rung 241
LD TIM123
OR TIM124
AND HR4.03
AND HR7.00
AND CNT013
LD HR5.06
ORNOT 61.00
LD HR6.00
ANDNOT 0.11
ANDNOT 0.12
AND 61.00
ORLD
ANDLD
DIFU(13) 10.06

